// TwinCAT 3 PLC project PLC
// ProgramVersion: 3.1.4023.0
// libraries:
//   Tc2_Standard, * (Beckhoff Automation GmbH)
//   Tc2_System, * (Beckhoff Automation GmbH)
//   Tc3_Module, * (Beckhoff Automation GmbH)
// project tree:
//   / PlcTask.TcTTO
//   POUs/ BFB_Trigger.TcPOU, MAIN.TcPOU
// real-time tasks:
//   TASK PlcTask: cycle T#10ms, priority 20, ADS port 350

CONFIGURATION PLC
    RESOURCE PLC ON TwinCAT3
        TASK PlcTask(INTERVAL := T#10ms, PRIORITY := 20);
        PROGRAM MAIN WITH PlcTask : MAIN;
    END_RESOURCE
END_CONFIGURATION

// ---- POUs/MAIN.TcPOU
PROGRAM MAIN
VAR
	fbTrig_Test				:BFB_Trigger;
	bTest					:BOOL;
	i						:INT;
	j						:INT;
END_VAR

fbTrig_Test(bIn := bTest);

IF fbTrig_Test.bRiseTrig THEN
	i := i + 1;
ELSIF fbTrig_Test.bFallTrig THEN
	i := i - 1;
END_IF

IF fbTrig_Test.bTrig THEN
	j := j + 1;
END_IF

END_PROGRAM

// ---- POUs/BFB_Trigger.TcPOU
(*-----------------------------------------版本信息-----------------------------------------
第一版本：		V1.0.0
功能说明：		边缘触发功能块集合
开发者：		Long.Yun
开发时间：		2021.09.02

变更版本：
版本			变更者		变更时间		变更说明
------------------------------------------------------------------------------------------*)
{attribute 'hide_all_locals'}
FUNCTION_BLOCK BFB_Trigger
VAR_INPUT
	//触发位
	bIn			:BOOL;
END_VAR

VAR_OUTPUT
	//边沿交替输出
	bTrig		:BOOL;
	//上升沿输出
	bRiseTrig	:BOOL;
	//下降沿输出
	bFallTrig	:BOOL;
END_VAR

VAR
	fbTrigR		:R_TRIG;
	fbTrigF		:F_TRIG;
END_VAR

fbTrigR(CLK := bIn, Q =>bRiseTrig);

fbTrigF(CLK := bIn, Q => bFallTrig);

bTrig := bRiseTrig OR bFallTrig;

END_FUNCTION_BLOCK
